FUNCTION_BLOCK FB_PPM_PowerMeter
VAR_INPUT
    fTempSP: REAL;
    bVetoTempFFO: BOOL;
    sDeviceName: STRING;

    // Used to know when to stop background auto-collection
    eEnumGet: E_PPM_States;
    stYAxisState: DWORD;

    // Calibrated for each gentec, should be passed as input
    // If not set, responsive energy will not be calculated
    {attribute 'pytmc' := '
        pv: RESP
        io: i
        field: EGU V/W
    '}
    fResponsivity: LREAL;

    // Passed to FB_AnalogInput
    // The initial values are correct for EL3062,
    // but not for EL3602, which needs iTermBits:=31
    // with fTermMax and fTermMin dependent on what
    // range the terminal was configured to use
    // (default -10000mV to +10000mV)
    iTermBits : UINT := 15;
    fTermMax : REAL := 10000;
    fTermMin: REAL := 0;
END_VAR
VAR_IN_OUT
    fbFFHWO: FB_HardwareFFOutput;
END_VAR
VAR
    iVoltageINT AT %I*: DINT;

    {attribute 'pytmc' := '
        pv: VOLT
        io: input
        field: EGU mV
    '}
    fVoltage: LREAL;

    {attribute 'pytmc' := '
        pv: VOLT_BUFFER
        io: input
        field: EGU mV
    '}
    fVoltageBuffer: ARRAY[1..1000] OF LREAL;

    {attribute 'pytmc' := '
        pv: STC
        io: input
    '}
    fbTempSensor: FB_CC_TempSensor;


    fFrequency: REAL;
    // Used to get beam rate
    {attribute 'pytmc' := '
        pv: SXR_NC_BeamRateFromEpics
        link: EVNT:SYS0:1:NC_SOFTRATE
    '}
    fSXR_NC_Frequency: REAL;
    {attribute 'pytmc' := '
        pv: SXR_SC_BeamRateFromEpics
        link: TPG:SYS0:1:DST04:RATE_RBV
    '}
    uSXR_SC_Frequency: UINT;

    {attribute 'pytmc' := '
        pv: HXR_NC_BeamRateFromEpics
        link: EVNT:SYS0:1:NC_HARDRATE
    '}
    fHXR_NC_Frequency: REAL;
    {attribute 'pytmc' := '
        pv: HXR_SC_BeamRateFromEpics
        link: TPG:SYS0:1:DST03:RATE_RBV
    '}
    uHXR_SC_Frequency: UINT;

    // Pulse-by-pulse energy and buffer
    {attribute 'pytmc' := '
        pv: MJ
        io: i
        field: EGU mJ
    '}
    fCalibMJ: LREAL;
    {attribute 'pytmc' := '
        pv: MJ_BUFFER
        io: i
        field: EGU mJ
    '}
    fCalibMJBuffer: ARRAY[1..1000] OF LREAL;

    // Wattage and buffer
    {attribute 'pytmc' := '
        pv: WATT
        io: i
        field: EGU mW
    '}
    fPulseWattage: LREAL;
    {attribute 'pytmc' := '
        pv: WATT_BUFFER
        io: i
        field: EGU mW
    '}
    fPulseWattageBuffer: ARRAY[1..1000] OF LREAL;

    // Background voltage
    {attribute 'pytmc' := '
        pv: BACK:VOLT
        io: io
        field: EGU mV
    '}
    fBackgroundVoltage: LREAL;

    // Internal variables for background voltage auto-collection
    fBackgroundVoltageAcc: LREAL;
    uAccCount: UINT;
    fBackgroundVoltageSum: LREAL;
    fBackgroundVoltageStale: LREAL;
    tonBackgroundAutoCollecting: TON;
    fBackgroundVoltageBuffer: ARRAY[1..100] OF LREAL;
    udBackgroundVoltageBufferIndex: UDINT := 1;
    rTrig_Background : R_TRIG;
    i: UDINT;
    // Used to reset auto-collected background buffer, and fBackgroundVoltage if in Auto mode
    {attribute 'pytmc' := '
        pv: BACK:RESET
        io: io
    '}
    bResetAutoBackground: BOOL;

    // In manual mode, auto-background updates buffer but does not change fBackgroundVoltage
    {attribute 'pytmc' := '
        pv: BACK:MODE
        io: io
    '}
    BACKGROUND_MODE: (Manual, Auto) := Auto;

    // Boolean to trigger collection of background voltages
    {attribute 'pytmc' := '
        pv: BACK:COLL
        io: io
    '}
    bBackgroundCollect: BOOL;

    // Time in seconds to collect background voltages for
    {attribute 'pytmc' := '
        pv: BACK:TIME
        io: io
        field: EGU s
    '}
    uBackgroundCollectionTime: UINT := 60;
    tofBackgroundCollecting: TOF;
    udBackgroundManualCount: UDINT;
    // Boolean indicating when background is being manually collected
    {attribute 'pytmc' := '
        pv: BACK:MANUAL_COLLECTING
        io: i
    '}
    bBackgroundCollecting: BOOL := FALSE;

    fbGetPMVoltage: FB_AnalogInput;

    fbVoltageBuffer: FB_LREALBuffer;
    fbPulseWattageBuffer: FB_LREALBuffer;
    fbCalibMJBuffer: FB_LREALBuffer;
END_VAR

fbTempSensor(
    fFaultThreshold:=fTempSP,
    bVeto:=bVetoTempFFO,
    sDevName:=sDeviceName,
    io_fbFFHWO:=fbFFHWO,
);

// Convert the terminal's integer into a value in millivolts
// If you get a compile-time error about converting type DINT
// to type INT, update your lcls-general version to at least
// v2.12.0
fbGetPMVoltage(
    iRaw := TO_INT(iVoltageINT),
    iTermBits := iTermBits,
    fTermMax := fTermMax,
    fTermMin := fTermMin,
    fReal => fVoltage);

rTrig_Background(CLK:=(eEnumGet <> E_PPM_States.OUT OR stYAxisState <> 0));
// Reset buffer and related variables
IF rTrig_Background.Q OR bResetAutoBackground THEN
    IF bResetAutoBackground THEN
        bResetAutoBackground := FALSE;
        IF BACKGROUND_MODE = Auto THEN
            fBackgroundVoltage := 0;
        END_IF
    ELSE
        // Dump 5s worth of readings
        IF udBackgroundVoltageBufferIndex > 6 THEN
            FOR i := (udBackgroundVoltageBufferIndex - 5) TO (udBackgroundVoltageBufferIndex - 1) DO
                fBackgroundVoltageSum := fBackgroundVoltageSum - fBackgroundVoltageBuffer[((i-1) MOD 100) + 1];
            END_FOR
            udBackgroundVoltageBufferIndex := udBackgroundVoltageBufferIndex - 5;
            IF udBackgroundVoltageBufferIndex <> 1 AND BACKGROUND_MODE = Auto THEN
                fBackgroundVoltage := fBackgroundVoltageSum / MIN((udBackgroundVoltageBufferIndex - 1), 100);
            END_IF
        ELSIF BACKGROUND_MODE = Auto THEN
                fBackgroundVoltage := 0;
        END_IF
    END_IF
    fBackgroundVoltageAcc := 0;
    fBackgroundVoltageSum := 0;
    tonBackgroundAutoCollecting(IN := FALSE);
    udBackgroundVoltageBufferIndex := 1;
ELSIF eEnumGet = E_PPM_States.OUT AND stYAxisState = 0 THEN
    tonBackgroundAutoCollecting( IN := TRUE, PT := T#1000MS);
    // Every second, move fBackgroundVoltageAcc into buffer and sum
    IF tonBackgroundAutoCollecting.Q = TRUE THEN
        tonBackgroundAutoCollecting( IN := FALSE);
        fBackgroundVoltageStale := fBackgroundVoltageBuffer[((udBackgroundVoltageBufferIndex - 1) MOD 100) + 1];
        fBackgroundVoltageBuffer[((udBackgroundVoltageBufferIndex - 1) MOD 100) + 1] := fBackgroundVoltageAcc / uAccCount;
        // Remove overwritten voltage
        IF udBackgroundVoltageBufferIndex > 100 THEN
            fBackgroundVoltageSum := fBackgroundVoltageSum - fBackgroundVoltageStale;
        END_IF
        fBackgroundVoltageSum := fBackgroundVoltageSum + fBackgroundVoltageAcc / uAccCount;
        fBackgroundVoltageAcc := fVoltage;
        uAccCount := 1;
        udBackgroundVoltageBufferIndex := udBackgroundVoltageBufferIndex + 1;
    ELSE
        uAccCount := uAccCount + 1;
        fBackgroundVoltageAcc := fBackgroundVoltageAcc + fVoltage;
    END_IF

END_IF

IF udBackgroundVoltageBufferIndex <> 1 AND BACKGROUND_MODE = Auto THEN
    fBackgroundVoltage := fBackgroundVoltageSum / MIN((udBackgroundVoltageBufferIndex - 1), 100);
END_IF

// Start collecting background in manual mode - 60s by default but can be set with uBackgroundCollectionTime
IF bBackgroundCollect = TRUE AND BACKGROUND_MODE = Manual THEN
    bBackgroundCollect := FALSE;
    udBackgroundManualCount := 0;
    fBackgroundVoltage := 0;
    tofBackgroundCollecting(IN := TRUE);
END_IF

bBackgroundCollecting := FALSE;
tofBackgroundCollecting(IN := FALSE, PT := UINT_TO_TIME(uBackgroundCollectionTime * 1000));
IF tofBackgroundCollecting.Q = TRUE THEN
    IF BACKGROUND_MODE = Manual THEN
        bBackgroundCollecting := TRUE;
        udBackgroundManualCount := udBackgroundManualCount + 1;
        fBackgroundVoltage := (fBackgroundVoltage * (udBackgroundManualCount - 1) + fVoltage) / udBackgroundManualCount;
    END_IF
END_IF

// Getting frequency based on accelerator source
{IF defined (K)}
    IF PMPS_GVL.stCurrentBeamParameters.nMachineMode = 0 THEN
        fFrequency := fSXR_NC_Frequency;
    ELSIF PMPS_GVL.stCurrentBeamParameters.nMachineMode = 1 THEN
        fFrequency := uSXR_SC_Frequency;
    END_IF
{ELSIF defined (L)}
    IF PMPS_GVL.stCurrentBeamParameters.nMachineMode = 0 THEN
        fFrequency := fHXR_NC_Frequency;
    ELSIF PMPS_GVL.stCurrentBeamParameters.nMachineMode = 1 THEN
        fFrequency := uHXR_SC_Frequency;
    END_IF
{END_IF}

// Getting wattage and energy
fPulseWattage := SEL(fResponsivity <> 0, 0, (fVoltage - fBackgroundVoltage) / fResponsivity);
fCalibMJ := SEL(fFrequency <> 0, -9999, fPulseWattage / fFrequency);

// Buffer the full-rate Voltage, Pulse wattage, and calibrated MJ values
fbVoltageBuffer(
    bExecute := TRUE,
    fInput := fVoltage,
    arrOutput => fVoltageBuffer);
fbPulseWattageBuffer(
    bExecute := TRUE,
    fInput := fPulseWattage,
    arrOutput => fPulseWattageBuffer);
fbCalibMJBuffer(
    bExecute := TRUE,
    fInput := fCalibMJ,
    arrOutput => fCalibMJBuffer);

END_FUNCTION_BLOCK

(* stored: Version 1.1.0.1
   POU FB_PPM_PowerMeter: Id {fedad4c7-7971-4466-a86d-d67d48d0e596}, SpecialFunc None *)
